INTERFACE I_StreamWriter

METHOD Add_BLOB : I_StreamWriter
VAR_INPUT
    Value : ANY;
END_VAR
END_METHOD

METHOD Add_BOOL : I_StreamWriter
VAR_INPUT
    Value : BOOL;
END_VAR
END_METHOD

METHOD Add_BYTE : I_StreamWriter
VAR_INPUT
    Value : BYTE;
END_VAR
END_METHOD

METHOD Add_DINT : I_StreamWriter
VAR_INPUT
    Value : DINT;
END_VAR
END_METHOD

METHOD Add_INT : I_StreamWriter
VAR_INPUT
    Value : INT;
END_VAR
END_METHOD

METHOD Add_LINT : I_StreamWriter
VAR_INPUT
    Value : LINT;
END_VAR
END_METHOD

METHOD Add_LREAL : I_StreamWriter
VAR_INPUT
    Value : LREAL;
END_VAR
END_METHOD

METHOD Add_PVOID : I_StreamWriter
VAR_INPUT
    Value : PVOID;
END_VAR
END_METHOD

METHOD Add_REAL : I_StreamWriter
VAR_INPUT
    Value : REAL;
END_VAR
END_METHOD

METHOD Add_STRING : I_StreamWriter
VAR_INPUT
    Value : STRING(255);
END_VAR
END_METHOD

METHOD Add_UDINT : I_StreamWriter
VAR_INPUT
    Value : UDINT;
END_VAR
END_METHOD

METHOD Add_UINT : I_StreamWriter
VAR_INPUT
    Value : UINT;
END_VAR
END_METHOD

METHOD Add_ULINT : I_StreamWriter
VAR_INPUT
    Value : ULINT;
END_VAR
END_METHOD

METHOD AppendBytesFromStream
VAR_INPUT
    StreamToAppend        : I_StreamReader;
    NumberOfBytesToAppend : UDINT;
END_VAR
VAR

END_VAR
END_METHOD

{attribute 'monitoring' := 'call'}
PROPERTY BufferAddress : PVOID
GET
END_GET
END_PROPERTY

METHOD Clear : I_StreamWriter
END_METHOD

METHOD Init
VAR_INPUT
    StreamLength : UDINT;
END_VAR
END_METHOD

{attribute 'monitoring' := 'call'}
PROPERTY ReadPosition : UDINT
GET
END_GET
END_PROPERTY

METHOD SetNextArgTypeId : I_StreamWriter
VAR_INPUT
    Value : E_ArgTypeId;
END_VAR
END_METHOD

METHOD SetReadPosition : I_StreamWriter
VAR_INPUT
    Position : UDINT;
END_VAR
END_METHOD

{attribute 'monitoring' := 'call'}
PROPERTY StreamLength : UDINT
GET
END_GET
END_PROPERTY

{attribute 'monitoring' := 'call'}
PROPERTY WritePosition : UDINT
GET
END_GET
END_PROPERTY

END_INTERFACE

(* stored: Version 1.1.0.1, ProductVersion 3.1.4024.9
   Itf I_StreamWriter: Id {ade11aac-fe77-01bf-2404-d979d6533839}
   Folder Methods: Id {a77095f2-d0ea-0978-3d8c-52df480fa7c6}
   Folder Properties: Id {bda3f685-2098-487c-8431-2b9eef1e7a95}
   Method Add_BLOB: Id {b462fbbf-cc66-4f5b-9718-73f4255ea87b}
   Method Add_BOOL: Id {8cf5fe7f-aa12-004e-3325-fcee77aea2e1}
   Method Add_BYTE: Id {1d7ff7ed-48e4-01a6-29b6-deba0ee3a148}
   Method Add_DINT: Id {0a63b2b6-3995-06e0-1f6f-61ea68a48505}
   Method Add_INT: Id {b8297403-f002-0df9-1bfd-5cbf1d20c6b5}
   Method Add_LINT: Id {ceecd414-20fc-0ffc-297e-96b5b4c79cb7}
   Method Add_LREAL: Id {c0904514-c94e-035d-2758-34432039059e}
   Method Add_PVOID: Id {9d72da79-66b0-056e-0951-45e0c7dba648}
   Method Add_REAL: Id {c7ce2c7d-2413-0856-0f2a-b4514e497708}
   Method Add_STRING: Id {7241d1d3-a603-0390-3368-f88e5b224128}
   Method Add_UDINT: Id {b1a663c4-27ab-0810-24ef-9325bfd028e7}
   Method Add_UINT: Id {ff28e4a5-26e3-0df4-04d0-5fe2f1d49971}
   Method Add_ULINT: Id {4d97bc5e-9e02-0fee-2770-fbac7ae79b7d}
   Method AppendBytesFromStream: Id {c441bda3-3b8a-4ed2-85ce-5e97568ff214}
   Property BufferAddress: Id {9bd5f99e-16ca-44bd-9ebe-71163e0cc2dc}
   Get Get: Id {38131e47-c458-48a0-b054-a51e7eacf53e}
   Method Clear: Id {dd7f97e5-7e5a-00e5-30c5-73909163ad6b}
   Method Init: Id {21f6d700-a942-4069-b090-b8315d873be7}
   Property ReadPosition: Id {000f0bc4-feb1-401f-8035-7c2f2ca24206}
   Get Get: Id {d90d4428-5495-4944-9bc4-d8654bdf7ca1}
   Method SetNextArgTypeId: Id {02a5322d-0101-4e1a-962e-ff0cf9820f93}
   Method SetReadPosition: Id {022de36b-fa7f-0b7c-1d93-83e7909f8ed3}
   Property StreamLength: Id {6dabb679-2ab6-4b83-89c1-6506b39d8105}
   Get Get: Id {ab50f728-0695-4ef2-8da7-1b25a7eed320}
   Property WritePosition: Id {8fd7c385-4e58-41ca-a924-76cab0827a45}
   Get Get: Id {001af59a-54e7-4229-aab2-3b48f26e187f} *)
